DATA_BLOCK "ST10_SafetyGate6_DB"
VAR
  "sSafetyGate Timer" : Array[1..5] of TON_TIME;
  sP_Trig : Array[1..10] of Bool;
  sN_Trig : Array[1..10] of Bool;
  "sSafetyGate UnlockRequest" : Bool;
  "sSafetyGate LockRequest" : Bool;
END_VAR
BEGIN
END_DATA_BLOCK
